//Enumeration for Machineunits
TYPE E_UnitName :
(
	eMachine		:= 1,
	eSample			:= 2
				
)DINT;
END_TYPE

(* stored: Version 1.1.0.1, ProductVersion 3.1.4024.12
   DUT E_UnitName: Id {38fb3a11-736e-4cc8-89e9-4c4bd7e49aca} *)
